FUNCTION_BLOCK SEL_DINT (* See SEL_ANY *)
  (* Standard: 61131-3 *)
  (* Version 0.1, 2006-09-14, JHC, Holobloc Inc, Converted to Template. *)
  (* Version 0.0, 2004-12-15, JHC, Rockwell Automation, Converted from SRC format. *)
  (* Compiler header: package fb.rt.plc.select; *)
  (* Compiler classdef: (G ? IN1 : IN0 ) *)
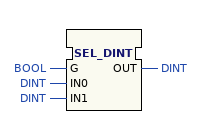
  VAR_INPUT
    G : BOOL;
    IN0 : DINT;
    IN1 : DINT;
  END_VAR
  VAR_OUTPUT
    OUT : DINT;
  END_VAR
END_FUNCTION_BLOCK
